// TIA Portal V20 export
FUNCTION "Flow_Sim" : Void   // FC14, FBD
{ S7_Optimized_Access := 'TRUE' }
// stored: SetENOAutomatically false
   VAR_TEMP
      Mul : Real;
      Dif : Real;
   END_VAR
BEGIN

REGION Network 1: flow value inlet
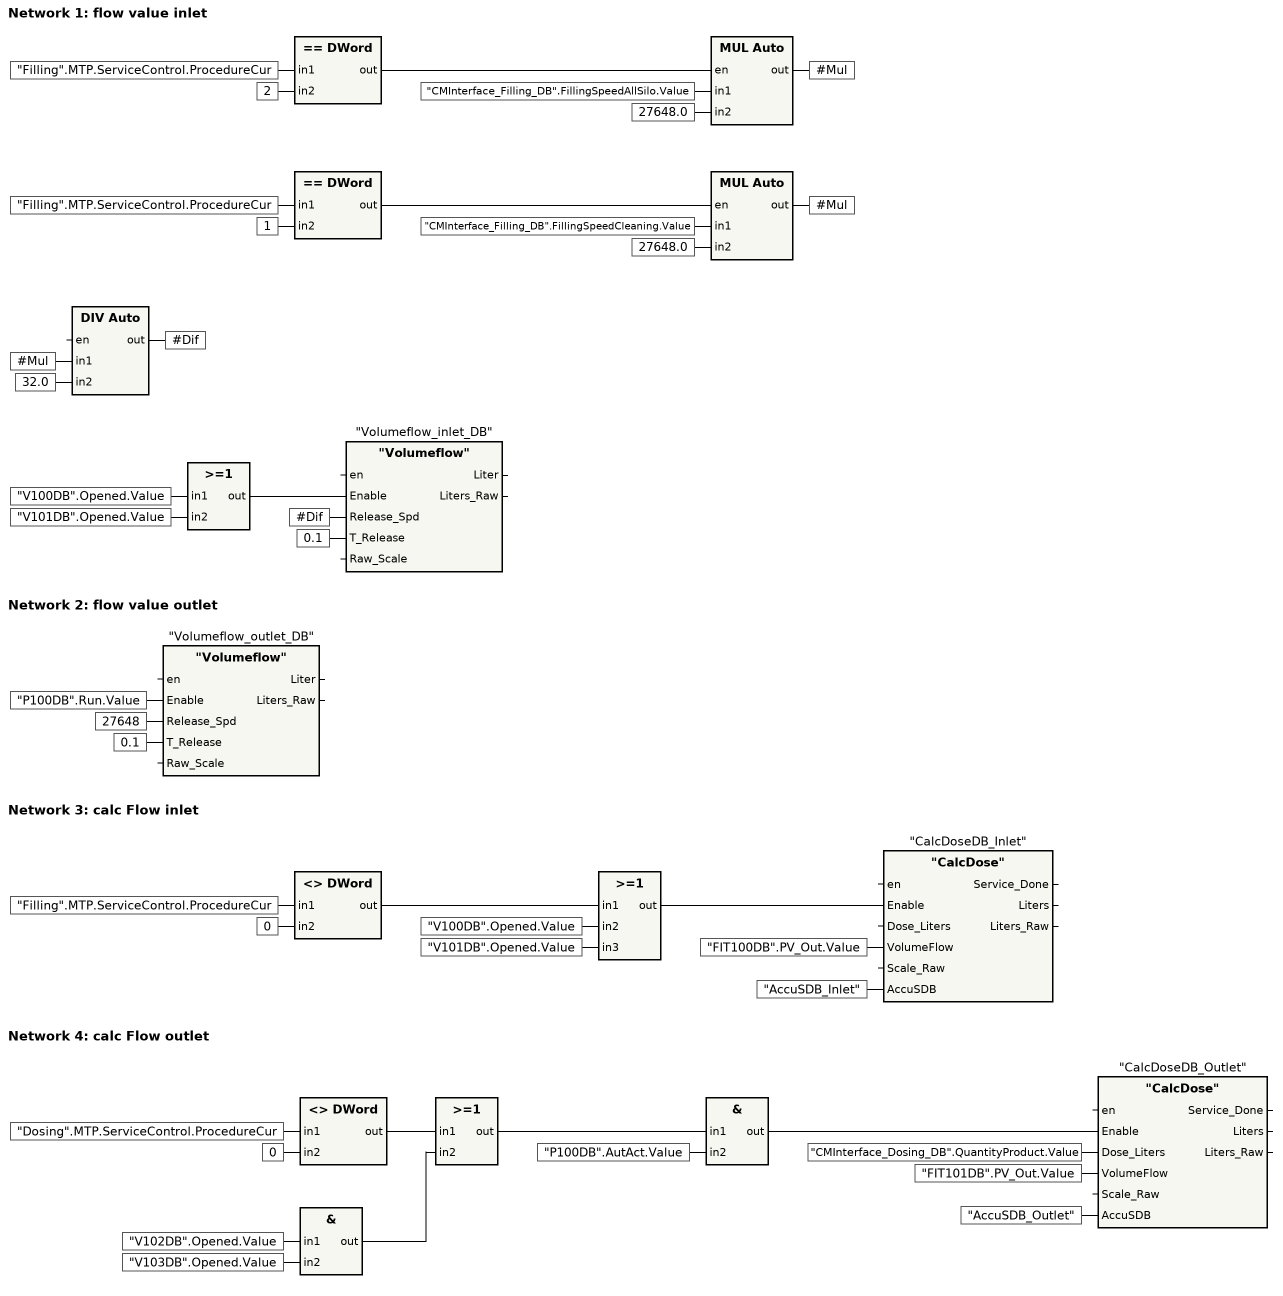
   IF "Filling".MTP.ServiceControl.ProcedureCur = 2 THEN
       #Mul := "CMInterface_Filling_DB".FillingSpeedAllSilo.Value * 27648.0;
   END_IF;
   IF "Filling".MTP.ServiceControl.ProcedureCur = 1 THEN
       #Mul := "CMInterface_Filling_DB".FillingSpeedCleaning.Value * 27648.0;
   END_IF;
   #Dif := #Mul / 32.0;
   "Volumeflow_inlet_DB"(Enable := "V100DB".Opened.Value OR "V101DB".Opened.Value,   // "Volumeflow"
                         Release_Spd := #Dif,
                         T_Release := 0.1);
END_REGION

REGION Network 2: flow value outlet
   "Volumeflow_outlet_DB"(Enable := "P100DB".Run.Value, Release_Spd := 27648, T_Release := 0.1);   // "Volumeflow"
END_REGION

REGION Network 3: calc Flow inlet
   "CalcDoseDB_Inlet"(Enable := ("Filling".MTP.ServiceControl.ProcedureCur <> 0) OR "V100DB".Opened.Value OR "V101DB".Opened.Value,   // "CalcDose"
                      VolumeFlow := "FIT100DB".PV_Out.Value,
                      AccuSDB := "AccuSDB_Inlet");
END_REGION

REGION Network 4: calc Flow outlet
   "CalcDoseDB_Outlet"(Enable := (("Dosing".MTP.ServiceControl.ProcedureCur <> 0) OR ("V102DB".Opened.Value AND "V103DB".Opened.Value)) AND "P100DB".AutAct.Value,   // "CalcDose"
                       Dose_Liters := "CMInterface_Dosing_DB".QuantityProduct.Value,
                       VolumeFlow := "FIT101DB".PV_Out.Value,
                       AccuSDB := "AccuSDB_Outlet");
END_REGION
END_FUNCTION
